{attribute 'qualified_only'}
{attribute 'strict'}
TYPE E_SCANNER_Vendor :
(
	SIEMENS		:= 1,
	MICROSCAN	:= 2,
	OMRON 		:= 3,
	KEYENCE		:= 4,
	COGNEX		:= 5
);
END_TYPE

(* stored: Version 1.1.0.1
   DUT E_SCANNER_Vendor: Id {83570167-cfb1-4910-a503-5d3eca7d19af} *)
